// TIA Portal V16 export
// export: Created 2024-06-24T15:42:27.8455031Z, ExportSetting WithDefaults, DisplayName Totally Integrated Automation Portal, DisplayVersion V16, DisplayName TIA Portal Version Control Interface, DisplayVersion V16, DisplayName TIA Portal Openness, DisplayVersion V16, DisplayName STEP 7 Professional, DisplayVersion V16, DisplayName STEP 7 Safety, DisplayVersion V16, DisplayName WinCC Advanced, DisplayVersion V16
FUNCTION_BLOCK "FB_WheelSorter"   // FB5, LAD
{ S7_Optimized_Access := 'TRUE' }
VERSION : 0.1
// stored: AutoNumber true, IsIECCheckEnabled false, IsRetainMemResEnabled false, MemoryReserve 100, SetENOAutomatically false, UDAEnableTagReadback false
   VAR_INPUT
      photoeyeEntry : Bool;
      photoeyeLeft : Bool;
      photoeyeRight : Bool;
      photoeyeStraight : Bool;
      machineReady : Bool;
   END_VAR
   VAR_OUTPUT
      beltConveyorLeft : Bool;
      beltConveyorRight : Bool;
      beltConveyorStraight : Bool;
      wheelSorterRight : Bool;
      wheelSorterStraight : Bool;
      wheelSorterLeft : Bool;
   END_VAR
   VAR_IN_OUT
      start : Bool;
      done : Bool;
      heavyLoad : Bool := false;
      lightLoad : Bool := false;
      mediumLoad : Bool := false;
   END_VAR
   VAR
      "step" : Array[0..20] of Bool;
   END_VAR
   VAR_TEMP   // added for the SCL form of the ladder/FBD networks
      _w1 : Bool;
      _w2 : Bool;
      _w3 : Bool;
   END_VAR
BEGIN

REGION Network 1
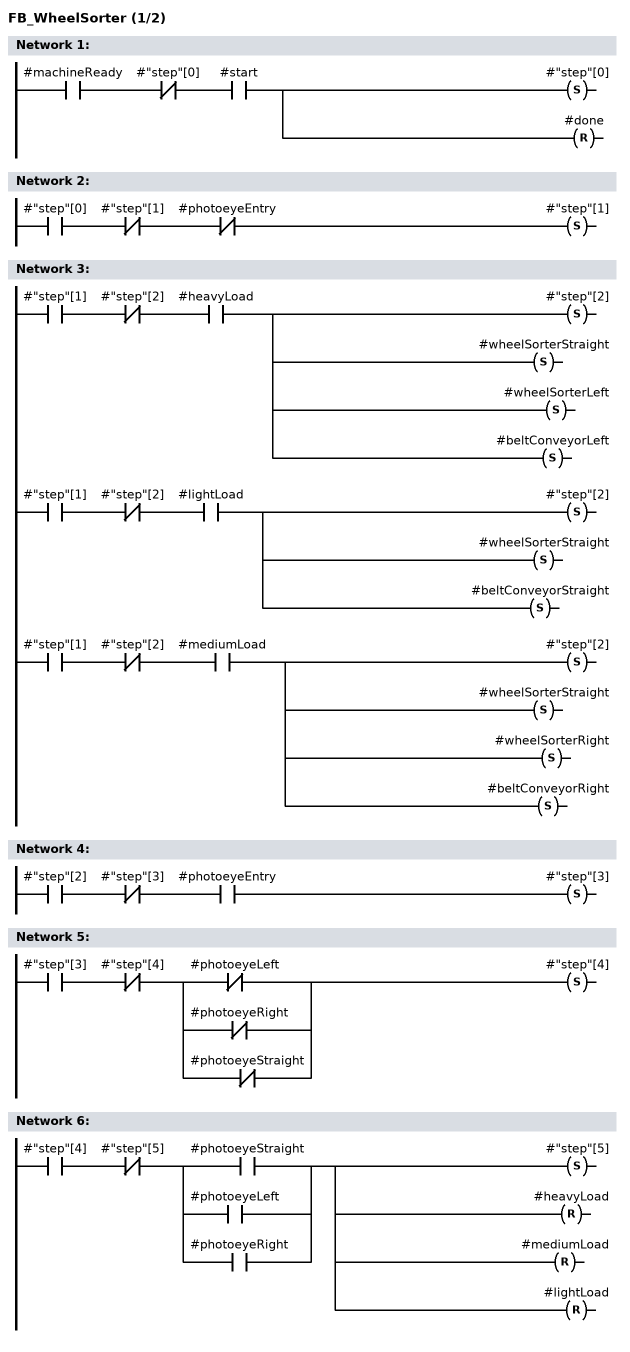
   RUNG wire#powerrail
      Contact( #machineReady )
      I_Contact( #"step"[0] )
      Contact( #start )
      wire#w1
      S_Coil( #"step"[0] )
   END_RUNG
   RUNG wire#w1
      R_Coil( #done )
   END_RUNG
   // the same network as SCL:
   #_w1 := #machineReady AND NOT #"step"[0] AND #start;
   IF #_w1 THEN
       #"step"[0] := TRUE;
       #done := FALSE;
   END_IF;
END_REGION

REGION Network 2
   RUNG wire#powerrail
      Contact( #"step"[0] )
      I_Contact( #"step"[1] )
      I_Contact( #photoeyeEntry )
      S_Coil( #"step"[1] )
   END_RUNG
   // the same network as SCL:
   IF #"step"[0] AND NOT #"step"[1] AND NOT #photoeyeEntry THEN #"step"[1] := TRUE; END_IF;
END_REGION

REGION Network 3
   RUNG wire#powerrail
      Contact( #"step"[1] )
      I_Contact( #"step"[2] )
      Contact( #heavyLoad )
      wire#w1
      S_Coil( #"step"[2] )
   END_RUNG
   RUNG wire#w1
      S_Coil( #wheelSorterStraight )
   END_RUNG
   RUNG wire#w1
      S_Coil( #wheelSorterLeft )
   END_RUNG
   RUNG wire#w1
      S_Coil( #beltConveyorLeft )
   END_RUNG
   RUNG wire#powerrail
      Contact( #"step"[1] )
      I_Contact( #"step"[2] )
      Contact( #lightLoad )
      wire#w2
      S_Coil( #"step"[2] )
   END_RUNG
   RUNG wire#w2
      S_Coil( #wheelSorterStraight )
   END_RUNG
   RUNG wire#w2
      S_Coil( #beltConveyorStraight )
   END_RUNG
   RUNG wire#powerrail
      Contact( #"step"[1] )
      I_Contact( #"step"[2] )
      Contact( #mediumLoad )
      wire#w3
      S_Coil( #"step"[2] )
   END_RUNG
   RUNG wire#w3
      S_Coil( #wheelSorterStraight )
   END_RUNG
   RUNG wire#w3
      S_Coil( #wheelSorterRight )
   END_RUNG
   RUNG wire#w3
      S_Coil( #beltConveyorRight )
   END_RUNG
   // the same network as SCL:
   #_w1 := #"step"[1] AND NOT #"step"[2] AND #heavyLoad;
   IF #_w1 THEN
       #"step"[2] := TRUE;
       #wheelSorterStraight := TRUE;
       #wheelSorterLeft := TRUE;
       #beltConveyorLeft := TRUE;
   END_IF;
   #_w2 := #"step"[1] AND NOT #"step"[2] AND #lightLoad;
   IF #_w2 THEN
       #"step"[2] := TRUE;
       #wheelSorterStraight := TRUE;
       #beltConveyorStraight := TRUE;
   END_IF;
   #_w3 := #"step"[1] AND NOT #"step"[2] AND #mediumLoad;
   IF #_w3 THEN
       #"step"[2] := TRUE;
       #wheelSorterStraight := TRUE;
       #wheelSorterRight := TRUE;
       #beltConveyorRight := TRUE;
   END_IF;
END_REGION

REGION Network 4
   RUNG wire#powerrail
      Contact( #"step"[2] )
      I_Contact( #"step"[3] )
      Contact( #photoeyeEntry )
      S_Coil( #"step"[3] )
   END_RUNG
   // the same network as SCL:
   IF #"step"[2] AND NOT #"step"[3] AND #photoeyeEntry THEN #"step"[3] := TRUE; END_IF;
END_REGION

REGION Network 5
   RUNG wire#powerrail
      Contact( #"step"[3] )
      I_Contact( #"step"[4] )
      wire#w1
      I_Contact( #photoeyeLeft )
      wire#w2
      S_Coil( #"step"[4] )
   END_RUNG
   RUNG wire#w1
      I_Contact( #photoeyeRight )
   END_RUNG wire#w2
   RUNG wire#w1
      I_Contact( #photoeyeStraight )
   END_RUNG wire#w2
   // the same network as SCL:
   IF #"step"[3] AND NOT #"step"[4] AND (NOT #photoeyeLeft OR NOT #photoeyeRight OR NOT #photoeyeStraight) THEN
       #"step"[4] := TRUE;
   END_IF;
END_REGION

REGION Network 6
   RUNG wire#powerrail
      Contact( #"step"[4] )
      I_Contact( #"step"[5] )
      wire#w1
      Contact( #photoeyeStraight )
      wire#w2
      S_Coil( #"step"[5] )
   END_RUNG
   RUNG wire#w1
      Contact( #photoeyeLeft )
   END_RUNG wire#w2
   RUNG wire#w1
      Contact( #photoeyeRight )
   END_RUNG wire#w2
   RUNG wire#w2
      R_Coil( #heavyLoad )
   END_RUNG
   RUNG wire#w2
      R_Coil( #mediumLoad )
   END_RUNG
   RUNG wire#w2
      R_Coil( #lightLoad )
   END_RUNG
   // the same network as SCL:
   #_w1 := #"step"[4] AND NOT #"step"[5] AND (#photoeyeStraight OR #photoeyeLeft OR #photoeyeRight);
   IF #_w1 THEN
       #"step"[5] := TRUE;
       #heavyLoad := FALSE;
       #mediumLoad := FALSE;
       #lightLoad := FALSE;
   END_IF;
END_REGION

REGION Network 7
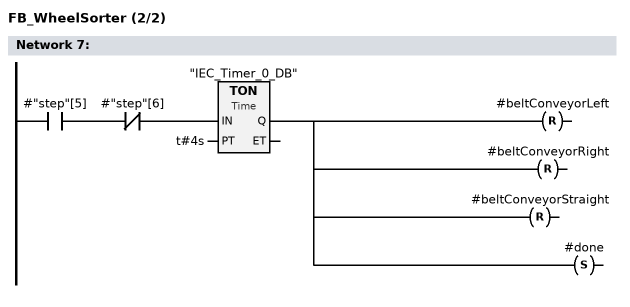
   RUNG wire#powerrail
      Contact( #"step"[5] )
      I_Contact( #"step"[6] )
      { S7_Templates := "time_type := Time" } "IEC_Timer_0_DB".TON(pt := t#4s, et =>)
      wire#w1
      R_Coil( #beltConveyorLeft )
   END_RUNG
   RUNG wire#w1
      R_Coil( #beltConveyorRight )
   END_RUNG
   RUNG wire#w1
      R_Coil( #beltConveyorStraight )
   END_RUNG
   RUNG wire#w1
      S_Coil( #done )
   END_RUNG
   // the same network as SCL:
   "IEC_Timer_0_DB".TON(IN := #"step"[5] AND NOT #"step"[6], PT := t#4s);
   IF "IEC_Timer_0_DB".Q THEN
       #beltConveyorLeft := FALSE;
       #beltConveyorRight := FALSE;
       #beltConveyorStraight := FALSE;
       #done := TRUE;
   END_IF;
END_REGION
END_FUNCTION_BLOCK
